// TIA Portal V19 export
FUNCTION "FC_FW_RES_QZ" : Void   // FC27, STL
TITLE = Reset Reserviertbits
{ S7_Optimized_Access := 'FALSE' }
AUTHOR : MS
// stored: AutoNumber false
   VAR_TEMP
      count : Int;
      DB_Nr : Int;
      B_PNTR : Int;
      newB_PNTR : Int;
      WT_DB : Int;
      adrRow : Int;
      WT_Nr : Int;
      WT_Nr_li : USInt;
      WT_Nr_re : USInt;
      Restzeit : Int;
      AdrPos : DWord;
      Pos : Byte;
      Pos2 : Byte;
      WT_Pos : USInt;
      Del_EndZiel : Bool;
      Ziel_belegt : Bool;
      amFW : Bool;
      AutoBef : Bool;
      no_UT_req : Bool;
      inA : Bool;
      outA : Bool;
      Sp_Bel : Bool;   // Speicher oder Beladepos
      ungerade : Bool;
      WT_Ziel_li : Int;
      WT_Ziel_re : Int;
   END_VAR
BEGIN

NETWORK
TITLE = Positionsdaten löschen
// Setz die Bits reservierte Quelle reserviertes ziel zurück
//------------------------------------
//Alles löschen
//------------------------------------
      SET;
      R     "DB_ANLAGE".IN.UT_Req;
      R     "DB_ANLAGE".OUT.WT_in_Anlage;
      L     0;
      T     "DB_ANLAGE".OUT.AnzUT_Req;

getP: L     "DB_ANLAGE".config.ANZ_Pos;
retP: T     #count;
      L     0;
      <=I;
      JC    dWT;
      L     #count;
      L     "DB_POS".LENG;
      *I;
      L     "DB_POS".Offset;
      +I;
      SLD   3;
      LAR1;
      OPN   "DB_POS";
      CLR;
      =     DBX [AR1, P#6.2];  //reserviert FW-Quelle
      =     DBX [AR1, P#6.3];  //reserviert FW-Ziel
      =     DBX [AR1, P#6.4];  //FW-kommt
      =     DBX [AR1, P#10.7];  //"DB_POS".POS[0].Checked

      L     0;  //Anlagenbad
      L     DBB [AR1, P#0.0];  //"DB_POS".POS[0].Typ
      <>I;
      A(;
      L     5;  //Speicherpos und Beladen zählt
      <=I;
      );
      =     #Sp_Bel;

      L     0;
      T     DBB [AR1, P#5.0];  //FW_Nr im Bad

      AN    DBX [AR1, P#96.0];  //"DB_POS".POS[0].belegt
      JC    setP;


      L     DBB [AR1, P#35.0];  //"DB_POS".POS[0].WT_DB
setP: T     DBB [AR1, P#36.0];  //"DB_POS".POS[0].next_WT


nexP: L     #count;
      LOOP  retP;

dWT:  L     "DB_ANLAGE".config.ANZ_WT;
reW:  T     #count;
      L     0;
      <=I;
      JC    endP;

      L     #count;
      +     100;
      T     #WT_DB;

//ungültige Position --> lösche WT_Nr_lang
      OPN   DB [#WT_DB];
      L     %DBB15;  //"DB_WT1".POS
      L     0;
      <>I;
      JC    WPok;
      T     %DBD6;  //"DB_WT1".WT_NR_lang

WPok: OPN   DB [#WT_DB];
      SET;
      R     %DBX20.6;  //"DB_WT1".noOPT_WT
      R     %DBX18.6;  //"DB_WT1".FW_Pos
      R     %DBX18.7;  //"DB_WT1".QT_Pos

      L     0;
      L     %DBD6;  //"DB_WT1".WT_NR_lang
      <>D;
      JC    WPos;
      L     %DBW2;  //"DB_WT1".OFFSET
      SLD   3;
      LAR1;
      L     0;
      T     DBD [AR1, P#0.0];  //Löschen erster Befehl
      T     DBD [AR1, P#4.0];
      T     %DBB36;  //"DB_WT1".End_Ziel_Pos
      T     %DBB37;  //"DB_WT1".End_Ziel_QT_Pos

WPos: L     0;
      L     %DBB36;  //"DB_WT1".End_Ziel_Pos
      ==I;
      R     %DBX20.5;  //"DB_WT1".noKorrBefx

      AN    "DB_ANLAGE".config.Anl_getaktet;
      JC    next;
      OPN   DB [#WT_DB];

      L     0;
      T     %DBB36;  //"DB_WT1".End_Ziel_Pos
      T     %DBB37;  //"DB_WT1".End_Ziel_QT_Pos

next: L     #count;
      LOOP  reW;

endP: NOP   0;

NETWORK
TITLE = Schleife über alle FW
// Positions- und WT-Informationen setzen

      L     0;
      T     #WT_Pos;

//------------------------------------
//WT-Nr laden und Bit amFW setzen
//------------------------------------
      OPN   DB [#DB_Nr];
      L     "DI_FW_1".ZST.WT_DB_NR_li;
      T     #WT_Nr_li;
      L     0;
      <>I;
      =     #amFW;

      L     "DI_FW_1".ZST.WT_DB_NR_re;
      T     #WT_Nr_re;
      L     0;
      <>I;
      S     #amFW;

      L     "DI_FW_1".ZST.BEFEHL.%B2;  //Befehlsart
      L     16#03;
      ==I;
      A     "DI_FW_1".ZST.Auto;
      =     #AutoBef;

      L     "DI_FW_1".ZST.Rest_Zeit;
      T     #Restzeit;

//FW hat WT aber keinen Befehl
// --> Daten aus WT holen und Quelle oder Ziel sperren
      A     #amFW;
      AN    #AutoBef;
      JC    SP_W;

//FW hat Befehl und WT bereits geholt
// --> WT aus Quelle holen und Quelle und Ziel sperren
      A     #amFW;
      A     #AutoBef;
      JC    SP_Z;

//FW hat Befehl aber WT noch nicht geholt
// --> WT aus Quelle holen und Quelle und Ziel sperren
      AN    #amFW;
      A     #AutoBef;
      JC    SP_Q;

//FW hat weder Befehl noch WT
// --> nächster FW
      JU    nexF;

//------------------------------------
//Quelle sperren
//------------------------------------
SP_Q: OPN   DB [#DB_Nr];
      L     0;
      L     "DI_FW_1".ZST.BEFEHL.%B1;  // Quelle
      ==I;
      JC    nexF;
      L     "DB_POS".LENG;
      *I;
      L     "DB_POS".Offset;
      +I;
      SLD   3;
      LAR1;

      L     "DI_FW_1".ZST.BEFEHL.%B1;  // Quelle
      L     2;
      MOD;
      A     <>0;
      =     #ungerade;

      OPN   "DB_POS";
      SET;
      S     DBX [AR1, P#6.2];  //reservierte Quelle

      L     DBB [AR1, P#35.0];  //WT_DB
      AN    #ungerade;
      JC    SP_Q_re;
      T     #WT_Nr_li;

      L     DBB [AR1, P#135.0];  //WT_DB
      <>I;
      JC    SP_Z;
      S     DBX [AR1, P#106.2];  //reservierte Quelle
SP_Q_re:T     #WT_Nr_re;
      JU    SP_Z;

//------------------------------------
//Ziel sperren
//------------------------------------
SP_Z: L     0;
      L     "DI_FW_1".ZST.BEFEHL.%B0;  // Ziel
      ==I;
      JC    nexF;
      L     2;
      MOD;
      A     <>0;
      L     "DI_FW_1".ZST.BEFEHL.%B0;  // Ziel
      JC    SP_Z_set;
      DEC   1;
SP_Z_set:T     #WT_Ziel_li;
      INC   1;
      T     #WT_Ziel_re;

SPWT: L     0;
      L     #WT_Ziel_li;
      ==I;
      JC    SPWT_re;
      L     "DB_POS".LENG;
      *I;
      L     "DB_POS".Offset;
      +I;
      SLD   3;
      LAR1;
      OPN   "DB_POS";
      SET;
      S     DBX [AR1, P#6.3];  //reserviertes Ziel

      L     0;
      L     #WT_Nr_li;
      >=I;
      JC    SPWT_re;

      OPN   "DB_POS";
      L     DBB [AR1, P#36.0];  //Next-WT
      L     0;
      <>I;
      JC    SPWT_re;

      L     #WT_Nr_li;
      T     DBB [AR1, P#36.0];  //Next-WT

      L     #WT_Nr_li;
      +     100;
      T     #WT_DB;

      OPN   DB [#WT_DB];
      SET;
      S     %DBX18.6;  //"DB_WT1".FW_Pos

SPWT_re:L     0;
      L     #WT_Ziel_re;
      ==I;
      JC    nexF;
      L     "DB_POS".LENG;
      *I;
      L     "DB_POS".Offset;
      +I;
      SLD   3;
      LAR1;
      OPN   "DB_POS";
      SET;
      S     DBX [AR1, P#6.3];  //reserviertes Ziel

      L     0;
      L     #WT_Nr_re;
      >=I;
      JC    nexF;

      OPN   "DB_POS";
      L     DBB [AR1, P#36.0];  //Next-WT
      L     0;
      <>I;
      JC    nexF;

      L     #WT_Nr_re;
      T     DBB [AR1, P#36.0];  //Next-WT

      L     #WT_Nr_re;
      +     100;
      T     #WT_DB;

      OPN   DB [#WT_DB];
      SET;
      S     %DBX18.6;  //"DB_WT1".FW_Pos

      JU    nexF;

//------------------------------------
//WT sperren
//------------------------------------
SP_W: L     0;
      T     #WT_Ziel_li;
      L     #WT_Nr_li;
      >=I;
      JC    SP_W_re;
      +     100;
      T     #WT_DB;

      OPN   DB [#WT_DB];
      L     0;
      L     %DBB21;  //"DB_WT1".Ziel_Pos_WT
      T     #WT_Ziel_li;
      <>I;
      JC    SP_W_re;
      L     %DBB15;
      T     #WT_Ziel_li;

SP_W_re:L     0;
      T     #WT_Ziel_re;
      L     #WT_Nr_re;
      >=I;
      JC    SPWT;
      +     100;
      T     #WT_DB;

      OPN   DB [#WT_DB];
      L     0;
      L     %DBB21;  //"DB_WT1".Ziel_Pos_WT
      T     #WT_Ziel_re;
      <>I;
      JC    SPWT;
      L     %DBB15;
      T     #WT_Ziel_re;
      JU    SPWT;

nexF: NOP   0;

endF: NOP   0;

NETWORK
TITLE = 
//------------------------------------
//WT kommt setzen
//------------------------------------
      L     "DB_ANLAGE".config.ANZ_WT;
retW: T     #count;
      L     0;
      <=I;
      JC    endW;

      L     #count;
      T     #WT_Nr;
      L     100;
      +I;
      T     #WT_DB;

//aktuellen Befehl auslesen
      OPN   DB [#WT_DB];
      L     0;
      L     %DBD6;  //"DB_WT1".WT_NR_lang
      ==D;
      T     %DBB62;  //"DB_WT1".akt_CMD
      JC    nexW;

      OPN   DB [#WT_DB];
      L     0;
      L     %DBB15;  //"DB_WT1".POS
      ==I;
      JC    nexW;
      L     %DBW48;  //"DB_WT1".B_PNTER
      L     %DBW4;  //"DB_WT1".LENG
      *D;
      L     %DBW2;  //"DB_WT1".OFFSET
      +D;
      SLD   3;
      LAR1;
      L     DBB [AR1, P#0.0];  //"DB_WT1".Befehl[x].Kennung
      T     %DBB62;  //"DB_WT1".akt_CMD

//------------------------------------
//DBB36 testen
//------------------------------------
Ncnt: OPN   DB [#WT_DB];
      A     %DBX18.6;  //"DB_WT1".FW_Pos
      O     %DBX18.7;  //"DB_WT1".QT_Pos
      JC    nexW;
      L     0;
      L     %DBB36;  //"DB_WT1".End_Ziel_Pos
      ==I;
      R     %DBX20.5;  //"DB_WT1".noKorrBefx
      JC    ckW;
      T     #WT_Pos;
      L     "DB_POS".LENG;
      *I;
      L     "DB_POS".Offset;
      +I;
      SLD   3;
      LAR1;
      OPN   "DB_POS";
      L     DBB [AR1, P#36.0];
      L     #WT_Nr;
      <>I;
      A(;
      L     DBB [AR1, P#36.0];
      L     0;
      <>I;
      );
      O(;
      L     DBB [AR1, P#0.0];  //PosTyp
      L     10;  //Typ QT
      <>I;
      A(;
      O     DBX [AR1, P#7.0];  //Sperre_in
      O     DBX [AR1, P#9.1];  //notFG_in
      );
      );
      JC    reSW;
      L     #WT_Nr;
      T     DBB [AR1, P#36.0];  //Next-WT

      CALL  "FC_FPosFree"
      ( WT_Nr    := #WT_Nr,
        Pos      := #WT_Pos,
        am_FW_QT := FALSE
      );
      JU    ckW;

reSW: OPN   DB [#WT_DB];
      L     0;
      T     %DBB36;

ckW:  L     0;
      L     %DBB15;  //"DB_WT1".POS
      ==I;
      JC    nexW;
      T     #WT_Pos;
      L     "DB_POS".LENG;
      *I;
      L     "DB_POS".Offset;
      +I;
      SLD   3;
      LAR1;
      OPN   "DB_POS";
      L     #count;
      L     DBB [AR1, P#35.0];
      ==I;
      AN    DBX [AR1, P#6.2];  //reserviert FW-Quelle
      AN    DBX [AR1, P#6.3];  //reserviert FW-Ziel
      AN    DBX [AR1, P#96.2];  //Vorruf
      AN    DBX [AR1, P#10.2];  //"DB_POS".POS[0].ignor_Exp
      A     DBX [AR1, P#6.0];  //Optipos
      A     DBX [AR1, P#6.1];  //berechnet
      JCN   ndel;
      OPN   DB [#WT_DB];
      L     0;
      T     %DBB36;  //"DB_WT1".End_Ziel_Pos
      T     %DBB37;  //"DB_WT1".End_Ziel_QT_Pos

ndel: OPN   "DB_POS";
      AN    DBX [AR1, P#9.3];  //FG_Posfree
      OPN   DB [#WT_DB];
      JC    nexW;

      CALL  "FC_FPosFree"
      ( WT_Nr    := #WT_Nr,
        Pos      := #WT_Pos,
        am_FW_QT := FALSE
      );

nexW: L     #count;
      LOOP  retW;

endW: NOP   0;
END_FUNCTION
